TYPE
    stSequenceTest :
    STRUCT
        WaitForStart   : INT := 10;
        OpenValveAandB : INT := 20;
    END_STRUCT
END_TYPE

(* stored: Version 1.1.0.1, ProductVersion 3.1.4024.12
   DUT stSequenceTest: Id {f2de1008-e973-410b-a43d-66735bffca97} *)
